# EPICS substitutions: NANODAC/NANODAC-IOC-01App/Db/nanodac.substitutions
file $(NANODAC)/db/nanodac.db
{
pattern {S, ND, NI}
	{\$(P),  "", 1}
}
